(* IEC 61131-3 sources: mect_apps/AnyTPAC/TestSuite/plc (part 3) *)

(* ---- or_P.st ---- *)
(*[[ ]]*)
PROGRAM or_P
#import "Crosstable.gvl"
#import "Resource1.gvl"
CONST
	this : int := 29;
	test_cases : int := 13;
END_CONST
VAR
	test_case : array [1..test_cases] of bit2_bit_T := [
		(input0 := 0, 		    input1 := 0, 	 	   ret_bool := 0, ret_byte := 0, 	 ret_word := 0, 	ret_dword := 0),
		(input0 := 0, 			input1 := 1, 	   	   ret_bool := 1, ret_byte := 1, 	 ret_word := 1, 	ret_dword := 1),
		(input0 := 1, 			input1 := 0, 	   	   ret_bool := 1, ret_byte := 1, 	 ret_word := 1, 	ret_dword := 1),
		(input0 := 1, 			input1 := 1, 	       ret_bool := 1, ret_byte := 1, 	 ret_word := 1, 	ret_dword := 1),
		(input0 := 0, 			input1 := 16#000000ff, ret_bool := 1, ret_byte := 16#ff, ret_word := 16#00ff, ret_dword := 16#000000ff),
		(input0 := 16#000000ff, input1 := 16#000000ff, ret_bool := 1, ret_byte := 16#ff, ret_word := 16#00ff, ret_dword := 16#000000ff),
		(input0 := 16#0000000f, input1 := 16#000000f0, ret_bool := 1, ret_byte := 16#ff, ret_word := 16#00ff, ret_dword := 16#000000ff),
		(input0 := 16#0000ffff, input1 := 16#0000ffff, ret_bool := 1, ret_byte := 16#ff, ret_word := 16#ffff, ret_dword := 16#0000ffff),
		(input0 := 16#0000ffff, input1 := 16#000000ff, ret_bool := 1, ret_byte := 16#ff, ret_word := 16#ffff, ret_dword := 16#0000ffff),
		(input0 := 16#0000f000, input1 := 16#0000ffff, ret_bool := 1, ret_byte := 16#ff, ret_word := 16#ffff, ret_dword := 16#0000ffff),
		(input0 := 16#000000ff, input1 := 16#0000ff00, ret_bool := 1, ret_byte := 16#ff, ret_word := 16#ffff, ret_dword := 16#0000ffff),
		(input0 := 16#abcde012, input1 := 16#ffffffff, ret_bool := 1, ret_byte := 16#ff, ret_word := 16#ffff, ret_dword := 16#ffffffff),
		(input0 := 16#abcdefab, input1 := 16#ff000000, ret_bool := 1, ret_byte := 16#ab, ret_word := 16#efab, ret_dword := 16#ffcdefab)
	];
    ret_bool   : bool;
    ret_byte   : byte;
    ret_word   : word;
    ret_dword  : dword;

	index : int := 1;
	expected : string;
	obtained : string;
	result : bool;
END_VAR

	if Status = STATUS_RUNNING AND test_level_29 > TEST_DISABLED and test_loops_29 < Target then

		(* ---------- test action ---------------*)
        ret_bool   := or(dword_to_bool(test_case[index].input0), dword_to_bool(test_case[index].input1));
        ret_byte   := or(dword_to_byte(test_case[index].input0), dword_to_byte(test_case[index].input1));
        ret_word   := or(dword_to_word(test_case[index].input0), dword_to_word(test_case[index].input1));
        ret_dword  := or(test_case[index].input0, test_case[index].input1);

		(* ---------- test condition ---------------*)
        result := (ret_bool = test_case[index].ret_bool)
		      and (ret_byte = test_case[index].ret_byte)
		      and (ret_word = test_case[index].ret_word)
		      and (ret_dword = test_case[index].ret_dword);

		(* ---------- log message ---------------*)
		expected := '';
		expected := CONCAT(expected, comma_blank, bool_to_string(test_case[index].ret_bool));
		expected := CONCAT(expected, comma_blank, byte_to_string(test_case[index].ret_byte));
		expected := CONCAT(expected, comma_blank, word_to_string(test_case[index].ret_word));
		expected := CONCAT(expected, comma_blank, dword_to_string(test_case[index].ret_dword));
		obtained := '';
		obtained := CONCAT(obtained, comma_blank, bool_to_string(ret_bool));
		obtained := CONCAT(obtained, comma_blank, byte_to_string(ret_byte));
		obtained := CONCAT(obtained, comma_blank, word_to_string(ret_word));
		obtained := CONCAT(obtained, comma_blank, dword_to_string(ret_dword));

		(* ---------- cycle ----------*)
		SingleTest(this, result, expected, obtained, test_cases,
				   index, test_level_29, test_counter_29, test_loops_29, test_errors_29);
	end_if;
END_PROGRAM

(* ---- pow_P.st ---- *)
(*[[ ]]*)
PROGRAM pow_P
#import "Crosstable.gvl"
#import "Resource1.gvl"
CONST
	this : int := 17;
	test_cases : int := 7;
	xl : lreal := 0.0000000000000001;
	x : real := 0.0000000000000001;
END_CONST
VAR
	test_case : array [1..test_cases] of lreal_lreal4_real4_T :=
[
(input:= 0.4487989505128276, retval1:=  1.5664296956520809, retval2:=-0.8011802632059132, retval3:=-0.3479481673201230, retval4:= 0.6699245856906788, retval5:=  1.5664297018771030, retval6:=-0.8011802543511257, retval7:=-0.3479481634745377, retval8:= 0.6699245886566987),
(input:= 0.8975979010256552, retval1:=  2.4537019914206710, retval2:=-0.1080330826459679, retval3:=-0.0469181716561418, retval4:= 0.9474164348509346, retval5:=  2.4537020109227896, retval6:=-0.1080330737911804, retval7:=-0.0469181678105565, retval8:= 0.9474164390455202),
(input:= 1.3463968515384828, retval1:=  3.8435516636419869, retval2:= 0.2974320254621965, retval3:= 0.1291730873995394, retval4:= 1.1603434196557856, retval5:=  3.8435514803715054, retval6:= 0.2974319900472387, retval7:= 0.1291730720190187, retval8:= 1.1603433991090293),
(input:= 1.7951958020513104, retval1:=  6.0206534627017669, retval2:= 0.5851140979139774, retval3:= 0.2541118240078394, retval4:= 1.3398491713813576, retval5:=  6.0206535584065408, retval6:= 0.5851141067687649, retval7:= 0.2541118278534247, retval8:= 1.3398491773133974),
(input:= 2.2439947525641379, retval1:=  9.4309303712065766, retval2:= 0.8082576492281872, retval3:= 0.3510218370158958, retval4:= 1.4979969134027407, retval5:=  9.4309299964728268, retval6:= 0.8082576315211277, retval7:= 0.3510218293258176, retval8:= 1.4979969001401805),
(input:= 2.6927937030769655, retval1:= 14.7728893910850854, retval2:= 0.9905792060221418, retval3:= 0.4302030830635206, retval4:= 1.6409734010875878, retval5:= 14.7728879822659920, retval6:= 0.9905791706071840, retval7:= 0.4302030676829999, retval8:= 1.6409733720300863),
(input:= 3.1415926535897931, retval1:= 23.1406926327792668, retval2:= 1.1447298858494002, retval3:= 0.4971498726941338, retval4:= 1.7724538509055159, retval5:= 23.1406946558030384, retval6:= 1.1447299136769349, retval7:= 0.4971498847794786, retval8:= 1.7724538755670267)
];
	input_lreal : lreal;
	input_real : real;
	retval1 : lreal;
	retval2 : lreal;
	retval3 : lreal;
	retval4 : lreal;
	retval5 : real;
	retval6 : real;
	retval7 : real;
	retval8 : real;

	index : int := 1;
	expected : string;
	obtained : string;
	result : bool;
END_VAR

	if Status = STATUS_RUNNING AND test_level_17 > TEST_DISABLED and test_loops_17 < Target then

		(* ---------- test action ---------------*)
		input_lreal := test_case[index].input;
		retval1 := exp(input_lreal);
		retval2 := ln(input_lreal);
		retval3 := log(input_lreal);
		retval4 := sqrt(input_lreal);
		input_real := lreal_to_real(test_case[index].input);
		retval5 := exp(input_real);
		retval6 := ln(input_real);
		retval7 := log(input_real);
		retval8 := sqrt(input_real);

		(* ---------- test condition ---------------*)
		result := (abs(retval1 - test_case[index].retval1) < xl)
		      and (abs(retval2 - test_case[index].retval2) < xl)
		      and (abs(retval3 - test_case[index].retval3) < xl)
		      and (abs(retval4 - test_case[index].retval4) < xl)
		      and (abs(retval5 - test_case[index].retval5) < x)
		      and (abs(retval6 - test_case[index].retval6) < x)
		      and (abs(retval7 - test_case[index].retval7) < x)
		      and (abs(retval8 - test_case[index].retval8) < x);

		(* ---------- log message ---------------*)
		expected := '';
		expected := CONCAT(expected, comma_blank, lreal_to_string(test_case[index].retval1));
		expected := CONCAT(expected, comma_blank, lreal_to_string(test_case[index].retval2));
		expected := CONCAT(expected, comma_blank, lreal_to_string(test_case[index].retval3));
		expected := CONCAT(expected, comma_blank, lreal_to_string(test_case[index].retval4));
		expected := CONCAT(expected, comma_blank, real_to_string(test_case[index].retval5));
		expected := CONCAT(expected, comma_blank, real_to_string(test_case[index].retval6));
		expected := CONCAT(expected, comma_blank, real_to_string(test_case[index].retval7));
		expected := CONCAT(expected, comma_blank, real_to_string(test_case[index].retval8));
		obtained := '';
		obtained := CONCAT(obtained, comma_blank, lreal_to_string(retval1));
		obtained := CONCAT(obtained, comma_blank, lreal_to_string(retval2));
		obtained := CONCAT(obtained, comma_blank, lreal_to_string(retval3));
		obtained := CONCAT(obtained, comma_blank, lreal_to_string(retval4));
		obtained := CONCAT(obtained, comma_blank, real_to_string(retval5));
		obtained := CONCAT(obtained, comma_blank, real_to_string(retval6));
		obtained := CONCAT(obtained, comma_blank, real_to_string(retval7));
		obtained := CONCAT(obtained, comma_blank, real_to_string(retval8));

		(* ---------- cycle ----------*)
		SingleTest(this, result, expected, obtained, test_cases,
				   index, test_level_17, test_counter_17, test_loops_17, test_errors_17);
	end_if;
END_PROGRAM

(* ---- real_to_all_P.st ---- *)
(*[[
]]*)
PROGRAM real_to_all_P
#import "Crosstable.gvl"
#import "Resource1.gvl"
CONST
	this : int := 7;
	test_cases : int := 5;
END_CONST
VAR
	test_case : array [1..test_cases] of real_all_T := [
		(input := 0.0, ret_bool := 0, ret_byte := 0, ret_dword := 0, ret_int := 0, ret_dint := 0, ret_lreal := 0.0,
		   ret_string := '0', ret_time := t#0ms, ret_udint := 0, ret_uint := 0, ret_word := 0),
		(input := 1.0, ret_bool := 1, ret_byte := 1, ret_dword := 1, ret_int := 1, ret_dint := 1, ret_lreal := 1.0,
		   ret_string := '1', ret_time := t#1ms, ret_udint := 1, ret_uint := 1, ret_word := 1),
		(input := -1.0, ret_bool := 1, ret_byte := 0, ret_dword := 0, ret_int := -1, ret_dint := -1, ret_lreal := -1.0,
		   ret_string := '-1', ret_time := t#-1ms, ret_udint := 0, ret_uint := 0, ret_word := 0),
		(input := 255.0, ret_bool := 1, ret_byte := 255, ret_dword := 255, ret_int := 255, ret_dint := 255, ret_lreal := 255.0,
		   ret_string := '255', ret_time := t#255ms, ret_udint := 255, ret_uint := 255, ret_word := 255),
		(input := 400.0, ret_bool := 1, ret_byte := 255, ret_dword := 400, ret_int := 400, ret_dint := 400, ret_lreal := 400.0,
		   ret_string := '400', ret_time := t#400ms, ret_udint := 400, ret_uint := 400, ret_word := 400)
	];
    ret_bool   : bool;
    ret_byte   : byte;
    ret_dword  : dword;
    ret_int    : int;
    ret_dint   : dint;
    ret_lreal  : lreal;
    ret_string : string;
	ret_time   : time;
    ret_udint  : udint;
    ret_uint   : uint;
    ret_word   : word;

	index : int := 1;
	expected : string;
	obtained : string;
	result : bool;
END_VAR

	if Status = STATUS_RUNNING AND test_level_07 > TEST_DISABLED and test_loops_07 < Target then

		(* ---------- test action ---------------*)
        ret_bool   := real_to_bool(test_case[index].input);
        ret_byte   := real_to_byte(test_case[index].input);
        ret_dword  := real_to_dword(test_case[index].input);
        ret_int    := real_to_int(test_case[index].input);
        ret_dint   := real_to_dint(test_case[index].input);
        ret_lreal  := real_to_lreal(test_case[index].input);
        ret_string := real_to_string(test_case[index].input);
        ret_time   := real_to_time(test_case[index].input);
        ret_udint  := real_to_udint(test_case[index].input);
        ret_uint   := real_to_uint(test_case[index].input);
        ret_word   := real_to_word(test_case[index].input);

		(* ---------- test condition ---------------*)
        result := (ret_bool = test_case[index].ret_bool)
		      and (ret_byte = test_case[index].ret_byte)
		      and (ret_dword = test_case[index].ret_dword)
		      and (ret_int = test_case[index].ret_int)
		      and (ret_dint = test_case[index].ret_dint)
		      and (ret_lreal = test_case[index].ret_lreal)
		      and (ret_string = test_case[index].ret_string)
		      and (ret_time = test_case[index].ret_time)
		      and (ret_udint = test_case[index].ret_udint)
		      and (ret_uint = test_case[index].ret_uint)
		      and (ret_word = test_case[index].ret_word);

		(* ---------- log message ---------------*)
		expected := '';
		expected := CONCAT(expected, comma_blank, bool_to_string(test_case[index].ret_bool));
		expected := CONCAT(expected, comma_blank, byte_to_string(test_case[index].ret_byte));
		expected := CONCAT(expected, comma_blank, dword_to_string(test_case[index].ret_dword));
		expected := CONCAT(expected, comma_blank, int_to_string(test_case[index].ret_int));
		expected := CONCAT(expected, comma_blank, dint_to_string(test_case[index].ret_dint));
		expected := CONCAT(expected, comma_blank, lreal_to_string(test_case[index].ret_lreal));
		expected := CONCAT(expected, comma_blank, test_case[index].ret_string);
		expected := CONCAT(expected, comma_blank, time_to_string(test_case[index].ret_time));
		expected := CONCAT(expected, comma_blank, udint_to_string(test_case[index].ret_udint));
		expected := CONCAT(expected, comma_blank, uint_to_string(test_case[index].ret_uint));
		expected := CONCAT(expected, comma_blank, word_to_string(test_case[index].ret_word));
		obtained := '';
		obtained := CONCAT(obtained, comma_blank, bool_to_string(ret_bool));
		obtained := CONCAT(obtained, comma_blank, byte_to_string(ret_byte));
		obtained := CONCAT(obtained, comma_blank, dword_to_string(ret_dword));
		obtained := CONCAT(obtained, comma_blank, int_to_string(ret_int));
		obtained := CONCAT(obtained, comma_blank, dint_to_string(ret_dint));
		obtained := CONCAT(obtained, comma_blank, lreal_to_string(ret_lreal));
		obtained := CONCAT(obtained, comma_blank, ret_string);
		obtained := CONCAT(obtained, comma_blank, time_to_string(ret_time));
		obtained := CONCAT(obtained, comma_blank, udint_to_string(ret_udint));
		obtained := CONCAT(obtained, comma_blank, uint_to_string(ret_uint));
		obtained := CONCAT(obtained, comma_blank, word_to_string(ret_word));

		(* ---------- cycle ----------*)
		SingleTest(this, result, expected, obtained, test_cases,
				   index, test_level_07, test_counter_07, test_loops_07, test_errors_07);
	end_if;

END_PROGRAM

(* ---- replace_P.st ---- *)
(*[[ ]]*)
PROGRAM replace_P
#import "Crosstable.gvl"
#import "Resource1.gvl"
CONST
	this : int := 49;
	test_cases : int := 3;
END_CONST
VAR
	test_case : array [1..test_cases] of string2_int2_string_T := [
		(input0 := 'stringa_dove_inserire', input1 := 'abc_', input2 := 4,  input3 := 1,  retval := 'abc_nga_dove_inserire'),
		(input0 := 'stringa_dove_inserire', input1 := 'abc_', input2 := 4,  input3 := 8,  retval := 'stringaabc_e_inserire'),
		(input0 := 'stringa_dove_inserire', input1 := 'abc_', input2 := 4,  input3 := 21, retval := 'stringa_dove_inserirabc_')
	];
    retval0   : string;
    retval1   : string;

	index : int := 1;
	expected : string;
	obtained : string;
	result : bool;
END_VAR

	if Status = STATUS_RUNNING AND test_level_49 > TEST_DISABLED and test_loops_49 < Target then

		(* ---------- test action ---------------*)
        retval0 := replace(test_case[index].input0, test_case[index].input1, test_case[index].input2, test_case[index].input3);
        retval1 := replace(test_case[index].input0, test_case[index].input1, int_to_dint(test_case[index].input2), int_to_dint(test_case[index].input3));

		(* ---------- test condition ---------------*)
        result := (retval0 = test_case[index].retval)
		      and (retval1 = test_case[index].retval);

		(* ---------- log message ---------------*)
		expected := '';
		expected := CONCAT(expected, comma_blank, test_case[index].retval);
		expected := CONCAT(expected, comma_blank, test_case[index].retval);
		obtained := '';
		obtained := CONCAT(obtained, comma_blank, retval0);
		obtained := CONCAT(obtained, comma_blank, retval1);

		(* ---------- cycle ----------*)
		SingleTest(this, result, expected, obtained, test_cases,
				   index, test_level_49, test_counter_49, test_loops_49, test_errors_49);
	end_if;
END_PROGRAM

(* ---- ro_P.st ---- *)
(*[[ ]]*)
PROGRAM ro_P (* gestisce sia rol che ror *)
#import "Crosstable.gvl"
#import "Resource1.gvl"
CONST
	this : int := 25;
	test_cases : int := 5;
END_CONST
VAR
	test_case : array [1..test_cases] of bit2_bit2_T := [
		(input0 := 16#abcdef11, input1 := 0, ret_bool := 1, ret_byte := 16#11, ret_word := 16#ef11, ret_dword := 16#abcdef11,
											 ret_bool2 := 1, ret_byte2 := 16#11, ret_word2 := 16#ef11, ret_dword2 := 16#abcdef11),
		(input0 := 16#abcdef11, input1 := 1, ret_bool := 1, ret_byte := 16#22, ret_word := 16#de23, ret_dword := 16#579bde23,
											 ret_bool2 := 1, ret_byte2 := 16#88, ret_word2 := 16#f788, ret_dword2 := 16#d5e6f788),
		(input0 := 16#abcdef12, input1 := 2, ret_bool := 1, ret_byte := 16#48, ret_word := 16#bc4b, ret_dword := 16#af37bc4a,
											 ret_bool2 := 1, ret_byte2 := 16#84, ret_word2 := 16#bbc4, ret_dword2 := 16#aaf37bc4),
		(input0 := 16#abcdef12, input1 := 4, ret_bool := 1, ret_byte := 16#21, ret_word := 16#f12e, ret_dword := 16#bcdef12a,
											 ret_bool2 := 1, ret_byte2 := 16#21, ret_word2 := 16#2ef1, ret_dword2 := 16#2abcdef1),
		(input0 := 16#abcdef12, input1 := 7, ret_bool := 1, ret_byte := 16#09, ret_word := 16#8977, ret_dword := 16#e6f78955,
											 ret_bool2 := 1, ret_byte2 := 16#24, ret_word2 := 16#25de, ret_dword2 := 16#25579bde)
	];
    ret_bool   : bool;
    ret_byte   : byte;
    ret_word   : word;
    ret_dword  : dword;
    ret_bool2  : bool;
    ret_byte2  : byte;
    ret_word2  : word;
    ret_dword2 : dword;

	index : int := 1;
	expected : string;
	obtained : string;
	result : bool;
END_VAR

	if Status = STATUS_RUNNING AND test_level_25 > TEST_DISABLED and test_loops_25 < Target then

		(* ---------- test action ---------------*)
        ret_bool   := rol(dword_to_bool(test_case[index].input0), dword_to_int(test_case[index].input1));
        ret_byte   := rol(dword_to_byte(test_case[index].input0), dword_to_int(test_case[index].input1));
        ret_word   := rol(dword_to_word(test_case[index].input0), dword_to_int(test_case[index].input1));
        ret_dword  := rol(test_case[index].input0, dword_to_int(test_case[index].input1));
        ret_bool2  := ror(dword_to_bool(test_case[index].input0), dword_to_int(test_case[index].input1));
        ret_byte2  := ror(dword_to_byte(test_case[index].input0), dword_to_int(test_case[index].input1));
        ret_word2  := ror(dword_to_word(test_case[index].input0), dword_to_int(test_case[index].input1));
        ret_dword2 := ror(test_case[index].input0, dword_to_int(test_case[index].input1));

		(* ---------- test condition ---------------*)
        result := (ret_bool = test_case[index].ret_bool)
		      and (ret_byte = test_case[index].ret_byte)
		      and (ret_word = test_case[index].ret_word)
		      and (ret_dword = test_case[index].ret_dword)
			  and (ret_bool2 = test_case[index].ret_bool2)
		      and (ret_byte2 = test_case[index].ret_byte2)
		      and (ret_word2 = test_case[index].ret_word2)
		      and (ret_dword2 = test_case[index].ret_dword2);

		(* ---------- log message ---------------*)
		expected := '';
		expected := CONCAT(expected, comma_blank, bool_to_string(test_case[index].ret_bool));
		expected := CONCAT(expected, comma_blank, byte_to_string(test_case[index].ret_byte));
		expected := CONCAT(expected, comma_blank, word_to_string(test_case[index].ret_word));
		expected := CONCAT(expected, comma_blank, dword_to_string(test_case[index].ret_dword));
		expected := CONCAT(expected, comma_blank, bool_to_string(test_case[index].ret_bool2));
		expected := CONCAT(expected, comma_blank, byte_to_string(test_case[index].ret_byte2));
		expected := CONCAT(expected, comma_blank, word_to_string(test_case[index].ret_word2));
		expected := CONCAT(expected, comma_blank, dword_to_string(test_case[index].ret_dword2));
		obtained := '';
		obtained := CONCAT(obtained, comma_blank, bool_to_string(ret_bool));
		obtained := CONCAT(obtained, comma_blank, byte_to_string(ret_byte));
		obtained := CONCAT(obtained, comma_blank, word_to_string(ret_word));
		obtained := CONCAT(obtained, comma_blank, dword_to_string(ret_dword));
		obtained := CONCAT(obtained, comma_blank, bool_to_string(ret_bool2));
		obtained := CONCAT(obtained, comma_blank, byte_to_string(ret_byte2));
		obtained := CONCAT(obtained, comma_blank, word_to_string(ret_word2));
		obtained := CONCAT(obtained, comma_blank, dword_to_string(ret_dword2));

		(* ---------- cycle ----------*)
		SingleTest(this, result, expected, obtained, test_cases,
				   index, test_level_25, test_counter_25, test_loops_25, test_errors_25);
	end_if;
END_PROGRAM

(* ---- rs_sr_P.st ---- *)
(*[[
]]*)
PROGRAM rs_sr_P
#import "Crosstable.gvl"
#import "Resource1.gvl"
CONST
	this : int := 52;
	test_cases : int := 11;
END_CONST
VAR
	test_case : array [1..test_cases] of bool2_bool2_T := [

		(input1 := false, input2 := false, retval1 := false, retval2 := false),
		(input1 := true,  input2 := false, retval1 := true,  retval2 := true),
		(input1 := false, input2 := false, retval1 := true,  retval2 := true),

		(input1 := false, input2 := false, retval1 := true,  retval2 := true),
		(input1 := false, input2 := true,  retval1 := false, retval2 := false),
		(input1 := false, input2 := false, retval1 := false, retval2 := false),

		(input1 := true,  input2 := true,  retval1 := false, retval2 := true),
		(input1 := false, input2 := false, retval1 := false, retval2 := true),
		(input1 := false, input2 := false, retval1 := false, retval2 := true),

		(input1 := false, input2 := true,  retval1 := false, retval2 := false),
		(input1 := false, input2 := false, retval1 := false, retval2 := false)
		];

    retval1  : bool;
    retval2  : bool;

	RS_Inst : RS;
	SR_Inst : SR;
	index : int := 1;
	expected : string;
	obtained : string;
	result : bool;
END_VAR

	if Status = STATUS_RUNNING AND test_level_52 > TEST_DISABLED and test_loops_52 < Target then

		(* ---------- test action ---------------*)
		RS_Inst(S := test_case[index].input1, R1 := test_case[index].input2, Q1 => retval1);
		SR_Inst(S1 := test_case[index].input1, R := test_case[index].input2, Q1 => retval2);

		(* ---------- test condition ---------------*)
        result := (retval1 = test_case[index].retval1)
		      and (retval2 = test_case[index].retval2);

		(* ---------- log message ---------------*)
		expected := '';
		expected := CONCAT(expected, comma_blank, bool_to_string(test_case[index].retval1));
		expected := CONCAT(expected, comma_blank, bool_to_string(test_case[index].retval2));
		obtained := '';
		obtained := CONCAT(obtained, comma_blank, bool_to_string(retval1));
		obtained := CONCAT(obtained, comma_blank, bool_to_string(retval2));

		(* ---------- cycle ----------*)
		SingleTest(this, result, expected, obtained, test_cases,
				   index, test_level_52, test_counter_52, test_loops_52, test_errors_52);
	end_if;
END_PROGRAM

(* ---- sel_P.st ---- *)
(*[[ ]]*)
PROGRAM sel_P
#import "Crosstable.gvl"
#import "Resource1.gvl"
CONST
	this : int := 35;
	test_cases : int := 2;
END_CONST
VAR
	test_case : array [1..test_cases] of bool_any2_any_T := [
		(input0 := false,  input1 := 20.0,  input2 := 30.0,  ret_byte := 20, ret_word := 20, ret_dword := 20, ret_int := 20, ret_dint := 20,
															ret_time := t#20ms, ret_real := 20.0, ret_lreal := 20.0, ret_string := '20'),
		(input0 := true,  input1 := 10.0,  input2 := 20.0,  ret_byte := 20, ret_word := 20, ret_dword := 20, ret_int := 20, ret_dint := 20,
															ret_time := t#20ms, ret_real := 20.0, ret_lreal := 20.0, ret_string := '20')
	];
    ret_byte   : byte;
    ret_word   : word;
    ret_dword  : dword;
    ret_int    : int;
    ret_dint   : dint;
    ret_time   : time;
    ret_real   : real;
    ret_lreal  : lreal;
    ret_string : string;

	index : int := 1;
	expected : string;
	obtained : string;
	result : bool;
END_VAR

	if Status = STATUS_RUNNING AND test_level_35 > TEST_DISABLED and test_loops_35 < Target then

		(* ---------- test action ---------------*)
        ret_byte    := sel(test_case[index].input0, lreal_to_byte(test_case[index].input1), lreal_to_byte(test_case[index].input2));
        ret_word    := sel(test_case[index].input0, lreal_to_word(test_case[index].input1), lreal_to_word(test_case[index].input2));
        ret_dword   := sel(test_case[index].input0, lreal_to_dword(test_case[index].input1), lreal_to_dword(test_case[index].input2));
        ret_int     := sel(test_case[index].input0, lreal_to_int(test_case[index].input1), lreal_to_int(test_case[index].input2));
        ret_dint    := sel(test_case[index].input0, lreal_to_dint(test_case[index].input1), lreal_to_dint(test_case[index].input2));
        ret_time    := sel(test_case[index].input0, lreal_to_time(test_case[index].input1), lreal_to_time(test_case[index].input2));
        ret_real    := sel(test_case[index].input0, lreal_to_real(test_case[index].input1), lreal_to_real(test_case[index].input2));
        ret_lreal   := sel(test_case[index].input0, test_case[index].input1, test_case[index].input2);
        ret_string  := sel(test_case[index].input0, lreal_to_string(test_case[index].input1), lreal_to_string(test_case[index].input2));

		(* ---------- test condition ---------------*)
        result := ((ret_byte = test_case[index].ret_byte)
			  and (ret_word = test_case[index].ret_word)
			  and (ret_dword = test_case[index].ret_dword)
			  and (ret_int = test_case[index].ret_int)
		      and (ret_dint = test_case[index].ret_dint)
		      and (ret_time = test_case[index].ret_time)
		      and (ret_real = test_case[index].ret_real)
		      and (ret_lreal = test_case[index].ret_lreal)
		      and (ret_string = test_case[index].ret_string));

		(* ---------- log message ---------------*)
		expected := '';
		expected := CONCAT(expected, comma_blank, byte_to_string(test_case[index].ret_byte));
		expected := CONCAT(expected, comma_blank, word_to_string(test_case[index].ret_word));
		expected := CONCAT(expected, comma_blank, dword_to_string(test_case[index].ret_dword));
		expected := CONCAT(expected, comma_blank, int_to_string(test_case[index].ret_int));
		expected := CONCAT(expected, comma_blank, dint_to_string(test_case[index].ret_dint));
		expected := CONCAT(expected, comma_blank, time_to_string(test_case[index].ret_time));
		expected := CONCAT(expected, comma_blank, real_to_string(test_case[index].ret_real));
		expected := CONCAT(expected, comma_blank, lreal_to_string(test_case[index].ret_lreal));
		expected := CONCAT(expected, comma_blank, test_case[index].ret_string);
		obtained := '';
		obtained := CONCAT(obtained, comma_blank, byte_to_string(ret_byte));
		obtained := CONCAT(obtained, comma_blank, word_to_string(ret_word));
		obtained := CONCAT(obtained, comma_blank, dword_to_string(ret_dword));
		obtained := CONCAT(obtained, comma_blank, int_to_string(ret_int));
		obtained := CONCAT(obtained, comma_blank, dint_to_string(ret_dint));
		obtained := CONCAT(obtained, comma_blank, time_to_string(ret_time));
		obtained := CONCAT(obtained, comma_blank, real_to_string(ret_real));
		obtained := CONCAT(obtained, comma_blank, lreal_to_string(ret_lreal));
		obtained := CONCAT(obtained, comma_blank, ret_string);

		(* ---------- cycle ----------*)
		SingleTest(this, result, expected, obtained, test_cases,
				   index, test_level_35, test_counter_35, test_loops_35, test_errors_35);
	end_if;
END_PROGRAM

(* ---- sh_P.st ---- *)
(*[[ ]]*)
PROGRAM sh_P (* gestisce sia shl che shr *)
#import "Crosstable.gvl"
#import "Resource1.gvl"
CONST
	this : int := 26;
	test_cases : int := 5;
END_CONST
VAR
	test_case : array [1..test_cases] of bit2_bit2_T := [
		(input0 := 16#abcdef11, input1 := 0, ret_bool := 1, ret_byte := 16#11, ret_word := 16#ef11, ret_dword := 16#abcdef11,
											 ret_bool2 := 1, ret_byte2 := 16#11, ret_word2 := 16#ef11, ret_dword2 := 16#abcdef11),
		(input0 := 16#abcdef11, input1 := 1, ret_bool := 0, ret_byte := 16#22, ret_word := 16#de22, ret_dword := 16#579bde22,
											 ret_bool2 := 0, ret_byte2 := 16#08, ret_word2 := 16#7788, ret_dword2 := 16#55e6f788),
		(input0 := 16#abcdef12, input1 := 2, ret_bool := 0, ret_byte := 16#48, ret_word := 16#bc48, ret_dword := 16#af37bc48,
											 ret_bool2 := 0, ret_byte2 := 16#04, ret_word2 := 16#3bc4, ret_dword2 := 16#2af37bc4),
		(input0 := 16#abcdef12, input1 := 4, ret_bool := 0, ret_byte := 16#20, ret_word := 16#f120, ret_dword := 16#bcdef120,
											 ret_bool2 := 0, ret_byte2 := 16#01, ret_word2 := 16#0ef1, ret_dword2 := 16#0abcdef1),
		(input0 := 16#abcdef12, input1 := 7, ret_bool := 0, ret_byte := 16#00, ret_word := 16#8900, ret_dword := 16#e6f78900,
											 ret_bool2 := 0, ret_byte2 := 16#00, ret_word2 := 16#01de, ret_dword2 := 16#01579bde)
	];
    ret_bool   : bool;
    ret_byte   : byte;
    ret_word   : word;
    ret_dword  : dword;
    ret_bool2  : bool;
    ret_byte2  : byte;
    ret_word2  : word;
    ret_dword2 : dword;

	index : int := 1;
	expected : string;
	obtained : string;
	result : bool;
END_VAR

	if Status = STATUS_RUNNING AND test_level_26 > TEST_DISABLED and test_loops_26 < Target then

		(* ---------- test action ---------------*)
        ret_bool   := shl(dword_to_bool(test_case[index].input0), dword_to_int(test_case[index].input1));
        ret_byte   := shl(dword_to_byte(test_case[index].input0), dword_to_int(test_case[index].input1));
        ret_word   := shl(dword_to_word(test_case[index].input0), dword_to_int(test_case[index].input1));
        ret_dword  := shl(test_case[index].input0, dword_to_int(test_case[index].input1));
        ret_bool2  := shr(dword_to_bool(test_case[index].input0), dword_to_int(test_case[index].input1));
        ret_byte2  := shr(dword_to_byte(test_case[index].input0), dword_to_int(test_case[index].input1));
        ret_word2  := shr(dword_to_word(test_case[index].input0), dword_to_int(test_case[index].input1));
        ret_dword2 := shr(test_case[index].input0, dword_to_int(test_case[index].input1));

		(* ---------- test condition ---------------*)
        result := (ret_bool = test_case[index].ret_bool)
		      and (ret_byte = test_case[index].ret_byte)
		      and (ret_word = test_case[index].ret_word)
		      and (ret_dword = test_case[index].ret_dword)
			  and (ret_bool2 = test_case[index].ret_bool2)
		      and (ret_byte2 = test_case[index].ret_byte2)
		      and (ret_word2 = test_case[index].ret_word2)
		      and (ret_dword2 = test_case[index].ret_dword2);

		(* ---------- log message ---------------*)
		expected := '';
		expected := CONCAT(expected, comma_blank, bool_to_string(test_case[index].ret_bool));
		expected := CONCAT(expected, comma_blank, byte_to_string(test_case[index].ret_byte));
		expected := CONCAT(expected, comma_blank, word_to_string(test_case[index].ret_word));
		expected := CONCAT(expected, comma_blank, dword_to_string(test_case[index].ret_dword));
		expected := CONCAT(expected, comma_blank, bool_to_string(test_case[index].ret_bool2));
		expected := CONCAT(expected, comma_blank, byte_to_string(test_case[index].ret_byte2));
		expected := CONCAT(expected, comma_blank, word_to_string(test_case[index].ret_word2));
		expected := CONCAT(expected, comma_blank, dword_to_string(test_case[index].ret_dword2));
		obtained := '';
		obtained := CONCAT(obtained, comma_blank, bool_to_string(ret_bool));
		obtained := CONCAT(obtained, comma_blank, byte_to_string(ret_byte));
		obtained := CONCAT(obtained, comma_blank, word_to_string(ret_word));
		obtained := CONCAT(obtained, comma_blank, dword_to_string(ret_dword));
		obtained := CONCAT(obtained, comma_blank, bool_to_string(ret_bool2));
		obtained := CONCAT(obtained, comma_blank, byte_to_string(ret_byte2));
		obtained := CONCAT(obtained, comma_blank, word_to_string(ret_word2));
		obtained := CONCAT(obtained, comma_blank, dword_to_string(ret_dword2));

		(* ---------- cycle ----------*)
		SingleTest(this, result, expected, obtained, test_cases,
				   index, test_level_26, test_counter_26, test_loops_26, test_errors_26);
	end_if;
END_PROGRAM

(* ---- string_to_all_P.st ---- *)
(*[[
]]*)
PROGRAM string_to_all_P
#import "Crosstable.gvl"
#import "Resource1.gvl"
CONST
	this : int := 8;
	test_cases : int := 5;
END_CONST
VAR
	test_case : array [1..test_cases] of string_all_T := [
		(input := '0', ret_bool := 0, ret_byte := 0, ret_dword := 0, ret_int := 0, ret_dint := 0, ret_lreal := 0.0,
		   ret_real := 0.0, ret_time := t#0ms, ret_udint := 0, ret_uint := 0, ret_word := 0),
		(input := '1', ret_bool := 1, ret_byte := 1, ret_dword := 1, ret_int := 1, ret_dint := 1, ret_lreal := 1.0,
		   ret_real := 1.0, ret_time := t#1ms, ret_udint := 1, ret_uint := 1, ret_word := 1),
		(input := '-1', ret_bool := 0, ret_byte := 255, ret_dword := 16#ffffffff, ret_int := -1, ret_dint := -1, ret_lreal := -1.0,
		   ret_real := -1.0, ret_time := t#-1ms, ret_udint := 16#ffffffff, ret_uint := 16#ffff, ret_word := 16#ffff),
		(input := '255', ret_bool := 0, ret_byte := 255, ret_dword := 255, ret_int := 255, ret_dint := 255, ret_lreal := 255.0,
		   ret_real := 255.0, ret_time := t#255ms, ret_udint := 255, ret_uint := 255, ret_word := 255),
		(input := '400', ret_bool := 0, ret_byte := 144, ret_dword := 400, ret_int := 400, ret_dint := 400, ret_lreal := 400.0,
		   ret_real := 400.0, ret_time := t#400ms, ret_udint := 400, ret_uint := 400, ret_word := 400)
	];
    ret_bool   : bool;
    ret_byte   : byte;
    ret_dword  : dword;
    ret_int    : int;
    ret_dint   : dint;
    ret_lreal  : lreal;
    ret_real   : real;
    ret_time   : time;
    ret_udint  : udint;
    ret_uint   : uint;
    ret_word   : word;

	index : int := 1;
	expected : string;
	obtained : string;
	result : bool;
END_VAR

	if Status = STATUS_RUNNING AND test_level_08 > TEST_DISABLED and test_loops_08 < Target then

		(* ---------- test action ---------------*)
        ret_bool   := string_to_bool(test_case[index].input);
        ret_byte   := string_to_byte(test_case[index].input);
        ret_dword  := string_to_dword(test_case[index].input);
        ret_int    := string_to_int(test_case[index].input);
        ret_dint   := string_to_dint(test_case[index].input);
        ret_lreal  := string_to_lreal(test_case[index].input);
        ret_real   := string_to_real(test_case[index].input);
        ret_time   := string_to_time(concat('t#', test_case[index].input, 'ms'));
        ret_udint  := string_to_udint(test_case[index].input);
        ret_uint   := string_to_uint(test_case[index].input);
        ret_word   := string_to_word(test_case[index].input);

		(* ---------- test condition ---------------*)
        result := (ret_bool = test_case[index].ret_bool)
		      and (ret_byte = test_case[index].ret_byte)
		      and (ret_dword = test_case[index].ret_dword)
		      and (ret_int = test_case[index].ret_int)
		      and (ret_dint = test_case[index].ret_dint)
		      and (ret_lreal = test_case[index].ret_lreal)
		      and (ret_real = test_case[index].ret_real)
		      and (ret_time = test_case[index].ret_time)
		      and (ret_udint = test_case[index].ret_udint)
		      and (ret_uint = test_case[index].ret_uint)
		      and (ret_word = test_case[index].ret_word);

		(* ---------- log message ---------------*)
		expected := '';
		expected := CONCAT(expected, comma_blank, bool_to_string(test_case[index].ret_bool));
		expected := CONCAT(expected, comma_blank, byte_to_string(test_case[index].ret_byte));
		expected := CONCAT(expected, comma_blank, dword_to_string(test_case[index].ret_dword));
		expected := CONCAT(expected, comma_blank, int_to_string(test_case[index].ret_int));
		expected := CONCAT(expected, comma_blank, dint_to_string(test_case[index].ret_dint));
		expected := CONCAT(expected, comma_blank, lreal_to_string(test_case[index].ret_lreal));
		expected := CONCAT(expected, comma_blank, real_to_string(test_case[index].ret_real));
		expected := CONCAT(expected, comma_blank, time_to_string(test_case[index].ret_time));
		expected := CONCAT(expected, comma_blank, udint_to_string(test_case[index].ret_udint));
		expected := CONCAT(expected, comma_blank, uint_to_string(test_case[index].ret_uint));
		expected := CONCAT(expected, comma_blank, word_to_string(test_case[index].ret_word));
		obtained := '';
		obtained := CONCAT(obtained, comma_blank, bool_to_string(ret_bool));
		obtained := CONCAT(obtained, comma_blank, byte_to_string(ret_byte));
		obtained := CONCAT(obtained, comma_blank, dword_to_string(ret_dword));
		obtained := CONCAT(obtained, comma_blank, int_to_string(ret_int));
		obtained := CONCAT(obtained, comma_blank, dint_to_string(ret_dint));
		obtained := CONCAT(obtained, comma_blank, lreal_to_string(ret_lreal));
		obtained := CONCAT(obtained, comma_blank, real_to_string(ret_real));
		obtained := CONCAT(obtained, comma_blank, time_to_string(ret_time));
		obtained := CONCAT(obtained, comma_blank, udint_to_string(ret_udint));
		obtained := CONCAT(obtained, comma_blank, uint_to_string(ret_uint));
		obtained := CONCAT(obtained, comma_blank, word_to_string(ret_word));

		(* ---------- cycle ----------*)
		SingleTest(this, result, expected, obtained, test_cases,
				   index, test_level_08, test_counter_08, test_loops_08, test_errors_08);
	end_if;

END_PROGRAM

(* ---- sub_P.st ---- *)
(*[[ ]]*)
PROGRAM sub_P
#import "Crosstable.gvl"
#import "Resource1.gvl"
CONST
	this : int := 24;
	test_cases : int := 4;
END_CONST
VAR
	test_case : array [1..test_cases] of num2_num_T := [
		(input0 := 10.0, input1 := 10.0, ret_int := 0, ret_dint := 0, ret_udint := 0, ret_uint := 0, ret_real := 0.0, ret_lreal := 0.0),
		(input0 := 10.0, input1 := 100.0, ret_int := -90, ret_dint := -90, ret_udint := 4294967206, ret_uint := 65446, ret_real := -90.0, ret_lreal := -90.0),
		(input0 := 100.0, input1 := 10.0, ret_int := 90, ret_dint := 90, ret_udint := 90, ret_uint := 90, ret_real := 90.0, ret_lreal := 90.0),
		(input0 := -10.0, input1 := -40.0, ret_int := 30, ret_dint := 30, ret_udint := 0, ret_uint := 0, ret_real := 30.0, ret_lreal := 30.0)
	];
    ret_int    : int;
    ret_dint   : dint;
    ret_uint   : uint;
    ret_udint  : udint;
    ret_real   : real;
    ret_lreal  : lreal;

	index : int := 1;
	expected : string;
	obtained : string;
	result : bool;
END_VAR

	if Status = STATUS_RUNNING AND test_level_24 > TEST_DISABLED and test_loops_24 < Target then

		(* ---------- test action ---------------*)
        ret_int     := sub(lreal_to_int(test_case[index].input0), lreal_to_int(test_case[index].input1));
        ret_dint    := sub(lreal_to_dint(test_case[index].input0), lreal_to_dint(test_case[index].input1));
        ret_uint    := sub(lreal_to_uint(test_case[index].input0), lreal_to_uint(test_case[index].input1));
        ret_udint   := sub(lreal_to_udint(test_case[index].input0), lreal_to_udint(test_case[index].input1));
        ret_real    := sub(lreal_to_real(test_case[index].input0), lreal_to_real(test_case[index].input1));
        ret_lreal   := sub(test_case[index].input0, test_case[index].input1);

		(* ---------- test condition ---------------*)
        result := ((ret_int = test_case[index].ret_int)
		      and (ret_dint = test_case[index].ret_dint)
		      and (ret_uint = test_case[index].ret_uint)
		      and (ret_udint = test_case[index].ret_udint)
		      and (ret_real = test_case[index].ret_real)
		      and (ret_lreal = test_case[index].ret_lreal));

		(* ---------- log message ---------------*)
		expected := '';
		expected := CONCAT(expected, comma_blank, int_to_string(test_case[index].ret_int));
		expected := CONCAT(expected, comma_blank, dint_to_string(test_case[index].ret_dint));
		expected := CONCAT(expected, comma_blank, uint_to_string(test_case[index].ret_uint));
		expected := CONCAT(expected, comma_blank, udint_to_string(test_case[index].ret_udint));
		expected := CONCAT(expected, comma_blank, real_to_string(test_case[index].ret_real));
		expected := CONCAT(expected, comma_blank, lreal_to_string(test_case[index].ret_lreal));
		obtained := '';
		obtained := CONCAT(obtained, comma_blank, int_to_string(ret_int));
		obtained := CONCAT(obtained, comma_blank, dint_to_string(ret_dint));
		obtained := CONCAT(obtained, comma_blank, uint_to_string(ret_uint));
		obtained := CONCAT(obtained, comma_blank, udint_to_string(ret_udint));
		obtained := CONCAT(obtained, comma_blank, real_to_string(ret_real));
		obtained := CONCAT(obtained, comma_blank, lreal_to_string(ret_lreal));

		(* ---------- cycle ----------*)
		SingleTest(this, result, expected, obtained, test_cases,
				   index, test_level_24, test_counter_24, test_loops_24, test_errors_24);
	end_if;
END_PROGRAM

(* ---- time_to_all_P.st ---- *)
(*[[
]]*)
PROGRAM time_to_all_P
#import "Crosstable.gvl"
#import "Resource1.gvl"
CONST
	this : int := 9;
	test_cases : int := 5;
END_CONST
VAR
	test_case : array [1..test_cases] of time_all_T := [
		(input := t#0ms, ret_dint := 0,  ret_int := 0, ret_lreal := 0.0, ret_real := 0.0, ret_string := 't#0ms'),
		(input := t#1ms, ret_dint := 1, ret_int := 1, ret_lreal := 1.0, ret_real := 1.0, ret_string := 't#1ms'),
		(input := t#-1ms, ret_dint := -1, ret_int := -1, ret_lreal := -1.0, ret_real := -1.0, ret_string := 't#-1ms'),
		(input := t#255ms, ret_dint := 255, ret_int := 255, ret_lreal := 255.0, ret_real := 255.0, ret_string := 't#255ms'),
		(input := t#400ms, ret_dint := 400, ret_int := 400, ret_lreal := 400.0, ret_real := 400.0, ret_string := 't#400ms')
	];
    ret_dint   : dint;
    ret_int    : int;
    ret_lreal  : lreal;
    ret_real   : real;
    ret_string : string;

	index : int := 1;
	expected: string;
	obtained: string;
	result : bool;
END_VAR

	if Status = STATUS_RUNNING AND test_level_09 > TEST_DISABLED and test_loops_09 < Target then

		(* ---------- test action ---------------*)
        ret_dint   := time_to_dint(test_case[index].input);
        ret_int    := time_to_int(test_case[index].input);
        ret_lreal  := time_to_lreal(test_case[index].input);
        ret_real   := time_to_real(test_case[index].input);
        ret_string := time_to_string(test_case[index].input);

		(* ---------- test condition ---------------*)
        result := (ret_dint = test_case[index].ret_dint)
		      and (ret_int = test_case[index].ret_int)
		      and (ret_lreal = test_case[index].ret_lreal)
		      and (ret_real = test_case[index].ret_real)
		      and (ret_string = test_case[index].ret_string);

		(* ---------- log message ---------------*)
		expected := '';
		expected := CONCAT(expected, comma_blank, dint_to_string(test_case[index].ret_dint));
		expected := CONCAT(expected, comma_blank, int_to_string(test_case[index].ret_int));
		expected := CONCAT(expected, comma_blank, lreal_to_string(test_case[index].ret_lreal));
		expected := CONCAT(expected, comma_blank, real_to_string(test_case[index].ret_real));
		expected := CONCAT(expected, comma_blank, test_case[index].ret_string);
		obtained := '';
		obtained := CONCAT(obtained, comma_blank, dint_to_string(ret_dint));
		obtained := CONCAT(obtained, comma_blank, int_to_string(ret_int));
		obtained := CONCAT(obtained, comma_blank, lreal_to_string(ret_lreal));
		obtained := CONCAT(obtained, comma_blank, real_to_string(ret_real));
		obtained := CONCAT(obtained, comma_blank, ret_string);

		(* ---------- cycle ----------*)
		SingleTest(this, result, expected, obtained, test_cases,
				   index, test_level_09, test_counter_09, test_loops_09, test_errors_09);
	end_if;
END_PROGRAM

(* ---- tof_ton_tp_P.st ---- *)
(*[[
]]*)
PROGRAM tof_ton_tp_P
#import "Crosstable.gvl"
#import "Resource1.gvl"
CONST
	this : int := 55;
	test_cases : int := 16;
END_CONST
VAR
	test_case : array [1..test_cases] of bool_time_bool3_time3_T := [

		(* reset all_____________________   TP______________________________  TON_____________________________  TOF_____________________________ *)
		(bool0 := false, time0 := t#000ms,  bool1 := false, time1 := t#000ms, bool2 := false, time2 := t#000ms, bool3 := false, time3 := t#000ms),

		(* start, reset TON, wait TP+TOF_   TP______________________________  TON_____________________________  TOF_____________________________ *)
		(bool0 := true,  time0 := t#250ms,  bool1 := true,  time1 := t#000ms, bool2 := false, time2 := t#000ms, bool3 := true,  time3 := t#000ms),
		(bool0 := false, time0 := t#250ms,  bool1 := true,  time1 := t#100ms, bool2 := false, time2 := t#000ms, bool3 := true,  time3 := t#000ms),
		(bool0 := false, time0 := t#250ms,  bool1 := true,  time1 := t#200ms, bool2 := false, time2 := t#000ms, bool3 := true,  time3 := t#100ms),
		(bool0 := false, time0 := t#250ms,  bool1 := false, time1 := t#000ms, bool2 := false, time2 := t#000ms, bool3 := true,  time3 := t#200ms),
		(bool0 := false, time0 := t#250ms,  bool1 := false, time1 := t#000ms, bool2 := false, time2 := t#000ms, bool3 := false, time3 := t#250ms),

		(* reset all_____________________   TP______________________________  TON_____________________________  TOF_____________________________ *)
		(bool0 := false, time0 := t#000ms,  bool1 := false, time1 := t#000ms, bool2 := false, time2 := t#000ms, bool3 := false, time3 := t#000ms),

		(* start and wait TP+TON_________   TP______________________________  TON_____________________________  TOF_____________________________ *)
		(bool0 := true,  time0 := t#250ms,  bool1 := true,  time1 := t#000ms, bool2 := false, time2 := t#000ms, bool3 := true,  time3 := t#000ms),
		(bool0 := true,  time0 := t#250ms,  bool1 := true,  time1 := t#100ms, bool2 := false, time2 := t#100ms, bool3 := true,  time3 := t#000ms),
		(bool0 := true,  time0 := t#250ms,  bool1 := true,  time1 := t#200ms, bool2 := false, time2 := t#200ms, bool3 := true,  time3 := t#000ms),
		(bool0 := true,  time0 := t#250ms,  bool1 := false, time1 := t#250ms, bool2 := true,  time2 := t#250ms, bool3 := true,  time3 := t#000ms),

		(* reset all_____________________   TP______________________________  TON_____________________________  TOF_____________________________ *)
		(bool0 := false, time0 := t#250ms,  bool1 := false, time1 := t#000ms, bool2 := false, time2 := t#000ms, bool3 := true,  time3 := t#000ms),

		(* start and wait TOF____________   TP______________________________  TON_____________________________  TOF_____________________________ *)
		(bool0 := false, time0 := t#250ms,  bool1 := false, time1 := t#000ms, bool2 := false, time2 := t#000ms, bool3 := true,  time3 := t#100ms),
		(bool0 := false, time0 := t#250ms,  bool1 := false, time1 := t#000ms, bool2 := false, time2 := t#000ms, bool3 := true,  time3 := t#200ms),
		(bool0 := false, time0 := t#250ms,  bool1 := false, time1 := t#000ms, bool2 := false, time2 := t#000ms, bool3 := false, time3 := t#250ms),

		(* reset all_____________________   TP______________________________  TON_____________________________  TOF_____________________________ *)
		(bool0 := false, time0 := t#000ms,  bool1 := false, time1 := t#000ms, bool2 := false, time2 := t#000ms, bool3 := false, time3 := t#000ms)
	];

    bool1, bool2, bool3 : bool;
    time1, time2, time3 : time;
	delta1, delta2, delta3: dint;

	TP_Inst : TP;
	TON_Inst : TON;
	TOF_Inst : TOF;
	index : int := 1;
	expected : string;
	obtained : string;
	result : bool;
	period_ms : time;
	info : tsk_info;
	retval : word;
END_VAR

	if Status = STATUS_RUNNING AND test_level_55 > TEST_DISABLED and test_loops_55 < Target then

		retval := TSK_GetInfo(TSK_GetMyName(), info);
		period_ms := info.tCycle;
		if period_ms <> t#100ms then
			MSG_SendToEng('ERROR: Program TOF_TON_TP must run @ 100ms: disabled.');
			test_level_55 := 0;
			return;
		end_if;

		(* ---------- test action ---------------*)
		TP_Inst (IN := test_case[index].bool0, PT := test_case[index].time0, Q => bool1, ET => time1);
		TON_Inst(IN := test_case[index].bool0, PT := test_case[index].time0, Q => bool2, ET => time2);
		TOF_Inst(IN := test_case[index].bool0, PT := test_case[index].time0, Q => bool3, ET => time3);

		delta1 := time_to_dint(time1 - test_case[index].time1);
		delta2 := time_to_dint(time2 - test_case[index].time2);
		delta3 := time_to_dint(time3 - test_case[index].time3);

		(* ---------- test condition ---------------*)
        result := (bool1 = test_case[index].bool1) and (abs(delta1) < 10)
		      and (bool2 = test_case[index].bool2) and (abs(delta2) < 10)
		      and (bool3 = test_case[index].bool3) and (abs(delta3) < 10);

		(* ---------- log message ---------------*)
		expected := '';
		expected := CONCAT(expected, comma_blank, bool_to_string(test_case[index].bool1));
		expected := CONCAT(expected, comma_blank, time_to_string(test_case[index].time1));
		expected := CONCAT(expected, comma_blank, bool_to_string(test_case[index].bool2));
		expected := CONCAT(expected, comma_blank, time_to_string(test_case[index].time2));
		expected := CONCAT(expected, comma_blank, bool_to_string(test_case[index].bool3));
		expected := CONCAT(expected, comma_blank, time_to_string(test_case[index].time3));
		obtained := '';
		obtained := CONCAT(obtained, comma_blank, bool_to_string(bool1));
		obtained := CONCAT(obtained, comma_blank, time_to_string(time1));
		obtained := CONCAT(obtained, comma_blank, bool_to_string(bool2));
		obtained := CONCAT(obtained, comma_blank, time_to_string(time2));
		obtained := CONCAT(obtained, comma_blank, bool_to_string(bool3));
		obtained := CONCAT(obtained, comma_blank, time_to_string(time3));

		(* ---------- cycle ----------*)
		if not result then
			;
		end_if;
		SingleTest(this, result, expected, obtained, test_cases,
				   index, test_level_55, test_counter_55, test_loops_55, test_errors_55);
	end_if;
END_PROGRAM

(* ---- trig_inv_P.st ---- *)
(*[[ ]]*)
PROGRAM trig_inv_P
#import "Crosstable.gvl"
#import "Resource1.gvl"
CONST
	this : int := 16;
	test_cases : int := 7;
	xl : lreal := 0.0000000000000010;
	x : real :=   0.0000000000000001;
END_CONST
VAR
	test_case : array [1..test_cases] of lreal_lreal3_real3_T :=
[
(input:= -1.0000000000000000, retval1:=-1.5707963267948966, retval2:= 3.1415926535897931, retval3:=-0.7853981633974483, retval4:=-1.5707963267948966, retval5:= 3.1415926535897931, retval6:=-0.7853981633974483),
(input:= -0.6666666666666667, retval1:=-0.7297276562269664, retval2:= 2.3005239830218631, retval3:=-0.5880026035475676, retval4:=-0.7297276828829742, retval5:= 2.3005240096778707, retval6:=-0.5880026173024855),
(input:= -0.3333333333333334, retval1:=-0.3398369094541220, retval2:= 1.9106332362490186, retval3:=-0.3217505543966422, retval4:=-0.3398369199908341, retval5:= 1.9106332467857308, retval6:=-0.3217505633373389),
(input:=  0.0000000000000000, retval1:= 0.0000000000000000, retval2:= 1.5707963267948966, retval3:= 0.0000000000000000, retval4:= 0.0000000000000000, retval5:= 1.5707963267948966, retval6:= 0.0000000000000000),
(input:=  0.3333333333333333, retval1:= 0.3398369094541219, retval2:= 1.2309594173407747, retval3:= 0.3217505543966421, retval4:= 0.3398369199908341, retval5:= 1.2309594068040626, retval6:= 0.3217505633373389),
(input:=  0.6666666666666665, retval1:= 0.7297276562269661, retval2:= 0.8410686705679304, retval3:= 0.5880026035475675, retval4:= 0.7297276828829742, retval5:= 0.8410686439119225, retval6:= 0.5880026173024855),
(input:=  1.0000000000000000, retval1:= 1.5707963267948966, retval2:= 0.0000000000000000, retval3:= 0.7853981633974483, retval4:= 1.5707963267948966, retval5:= 0.0000000000000000, retval6:= 0.7853981633974483)
];
	input_lreal : lreal;
	input_real : real;
	retval1 : lreal;
	retval2 : lreal;
	retval3 : lreal;
	retval4 : real;
	retval5 : real;
	retval6 : real;

	index : int := 1;
	expected : string;
	obtained : string;
	result : bool;
END_VAR

	if Status = STATUS_RUNNING AND test_level_16 > TEST_DISABLED and test_loops_16 < Target then

		(* ---------- test action ---------------*)
		input_lreal := test_case[index].input;
        retval1 := asin(input_lreal);
        retval2 := acos(input_lreal);
        retval3 := atan(input_lreal);
		input_real := lreal_to_real(test_case[index].input);
        retval4 := asin(input_real);
        retval5 := acos(input_real);
        retval6 := atan(input_real);

		(* ---------- test condition ---------------*)
        result := (abs(retval1 - test_case[index].retval1) < xl)
		      and (abs(retval2 - test_case[index].retval2) < xl)
		      and (abs(retval3 - test_case[index].retval3) < xl)
		      and (abs(retval4 - test_case[index].retval4) < x)
		      and (abs(retval5 - test_case[index].retval5) < x)
		      and (abs(retval6 - test_case[index].retval6) < x);

		(* ---------- log message ---------------*)
		expected := '';
		expected := CONCAT(expected, comma_blank, lreal_to_string(test_case[index].retval1));
		expected := CONCAT(expected, comma_blank, lreal_to_string(test_case[index].retval2));
		expected := CONCAT(expected, comma_blank, lreal_to_string(test_case[index].retval3));
		expected := CONCAT(expected, comma_blank, real_to_string(test_case[index].retval4));
		expected := CONCAT(expected, comma_blank, real_to_string(test_case[index].retval5));
		expected := CONCAT(expected, comma_blank, real_to_string(test_case[index].retval6));
		obtained := '';
		obtained := CONCAT(obtained, comma_blank, lreal_to_string(retval1));
		obtained := CONCAT(obtained, comma_blank, lreal_to_string(retval2));
		obtained := CONCAT(obtained, comma_blank, lreal_to_string(retval3));
		obtained := CONCAT(obtained, comma_blank, real_to_string(retval4));
		obtained := CONCAT(obtained, comma_blank, real_to_string(retval5));
		obtained := CONCAT(obtained, comma_blank, real_to_string(retval6));

		(* ---------- cycle ----------*)
		SingleTest(this, result, expected, obtained, test_cases,
				   index, test_level_16, test_counter_16, test_loops_16, test_errors_16);
	end_if;
END_PROGRAM

(* ---- trig_P.st ---- *)
(*[[ ]]*)
PROGRAM trig_P
#import "Crosstable.gvl"
#import "Resource1.gvl"
CONST
	this : int := 15;
	test_cases : int := 7;
	xl : lreal := 0.0000000000000001;
	x : real := 0.0000000000000001;
END_CONST
VAR
	test_case : array [1..test_cases] of lreal_lreal3_real3_T :=
[
(input:= 0.0000000000000000, retval1:= 0.0000000000000000, retval2:= 1.0000000000000000, retval3:= 0.0000000000000000, retval4:= 0.0000000000000000, retval5:= 1.0000000000000000, retval6:= 0.0000000000000000),
(input:= 1.0471975511965976, retval1:= 0.8660254037844386, retval2:= 0.5000000000000001, retval3:= 1.7320508075688767, retval4:= 0.8660254183549017, retval5:= 0.4999999747632170, retval6:= 1.7320509241325899),
(input:= 2.0943951023931953, retval1:= 0.8660254037844387, retval2:=-0.4999999999999998, retval3:=-1.7320508075688783, retval4:= 0.8660253746435105, retval5:=-0.5000000504735648, retval6:=-1.7320505744414876),
(input:= 3.1415926535897931, retval1:= 0.0000000000000001, retval2:=-1.0000000000000000, retval3:=-0.0000000000000001, retval4:=-0.0000000874227800, retval5:=-0.9999999999999962, retval6:= 0.0000000874227800),
(input:= 4.1887902047863905, retval1:=-0.8660254037844384, retval2:=-0.5000000000000004, retval3:= 1.7320508075688754, retval4:=-0.8660254620662861, retval5:=-0.4999998990528655, retval6:= 1.7320512738237981),
(input:= 5.2359877559829879, retval1:=-0.8660254037844390, retval2:= 0.4999999999999993, retval3:=-1.7320508075688805, retval4:=-0.8660254501414079, retval5:= 0.4999999197073655, retval6:=-1.7320511784247199),
(input:= 6.2831853071795862, retval1:=-0.0000000000000002, retval2:= 1.0000000000000000, retval3:=-0.0000000000000002, retval4:= 0.0000001748455600, retval5:= 0.9999999999999847, retval6:= 0.0000001748455600)
];
	input_lreal : lreal;
	input_real : real;
	retval1 : lreal;
	retval2 : lreal;
	retval3 : lreal;
	retval4 : real;
	retval5 : real;
	retval6 : real;

	index : int := 1;
	expected : string;
	obtained : string;
	result : bool;
END_VAR

	if Status = STATUS_RUNNING AND test_level_15 > TEST_DISABLED and test_loops_15 < Target then

		(* ---------- test action ---------------*)
		input_lreal := test_case[index].input;
        retval1 := sin(input_lreal);
        retval2 := cos(input_lreal);
        retval3 := tan(input_lreal);
		input_real := lreal_to_real(test_case[index].input);
        retval4 := sin(input_real);
        retval5 := cos(input_real);
        retval6 := tan(input_real);

		(* ---------- test condition ---------------*)
        result := (abs(retval1 - test_case[index].retval1) < xl)
		      and (abs(retval2 - test_case[index].retval2) < xl)
		      and (abs(retval3 - test_case[index].retval3) < xl)
		      and (abs(retval4 - test_case[index].retval4) < x)
		      and (abs(retval5 - test_case[index].retval5) < x)
		      and (abs(retval6 - test_case[index].retval6) < x);

		(* ---------- log message ---------------*)
		expected := '';
		expected := CONCAT(expected, comma_blank, lreal_to_string(test_case[index].retval1));
		expected := CONCAT(expected, comma_blank, lreal_to_string(test_case[index].retval2));
		expected := CONCAT(expected, comma_blank, lreal_to_string(test_case[index].retval3));
		expected := CONCAT(expected, comma_blank, real_to_string(test_case[index].retval4));
		expected := CONCAT(expected, comma_blank, real_to_string(test_case[index].retval5));
		expected := CONCAT(expected, comma_blank, real_to_string(test_case[index].retval6));
		obtained := '';
		obtained := CONCAT(obtained, comma_blank, lreal_to_string(retval1));
		obtained := CONCAT(obtained, comma_blank, lreal_to_string(retval2));
		obtained := CONCAT(obtained, comma_blank, lreal_to_string(retval3));
		obtained := CONCAT(obtained, comma_blank, real_to_string(retval4));
		obtained := CONCAT(obtained, comma_blank, real_to_string(retval5));
		obtained := CONCAT(obtained, comma_blank, real_to_string(retval6));

		(* ---------- cycle ----------*)
		SingleTest(this, result, expected, obtained, test_cases,
				   index, test_level_15, test_counter_15, test_loops_15, test_errors_15);
	end_if;
END_PROGRAM

(* ---- trunc_P.st ---- *)
(*[[
]]*)
PROGRAM trunc_P
#import "Crosstable.gvl"
#import "Resource1.gvl"
CONST
	this : int := 10;
	test_cases : int := 5;
END_CONST
VAR
	test_case : array [1..test_cases] of lreal_any_int_T := [
		(input := -7.0, ret_int :=  -7, ret_dint := -7),
		(input := -2.2, ret_int :=  -2, ret_dint := -2),
		(input := 14.0, ret_int := 14, ret_dint := 14),
		(input := 14.11, ret_int := 14, ret_dint := 14),
		(input := 14.88, ret_int := 14, ret_dint := 14)
	];
	ret_int1  : int;
	ret_int2  : int;
	ret_dint1 : dint;
	ret_dint2 : dint;

	index : int := 1;
	expected : string;
	obtained : string;
	result : bool;
END_VAR

	if Status = STATUS_RUNNING AND test_level_10 > TEST_DISABLED and test_loops_10 < Target then

		(* ---------- test action ---------------*)
        ret_int1  := trunc(test_case[index].input);
        ret_dint1 := trunc(test_case[index].input);
        ret_int2  := trunc(lreal_to_real(test_case[index].input));
        ret_dint2 := trunc(lreal_to_real(test_case[index].input));

		(* ---------- test condition ---------------*)
        result := (ret_int1 = test_case[index].ret_int)
				  and (ret_dint1 = test_case[index].ret_dint)
				  and (ret_int2 = test_case[index].ret_int)
				  and (ret_dint2 = test_case[index].ret_dint);

		(* ---------- log message ---------------*)
		expected := '';
		expected := CONCAT(expected, comma_blank, int_to_string(test_case[index].ret_int));
		expected := CONCAT(expected, comma_blank, int_to_string(test_case[index].ret_int));
		expected := CONCAT(expected, comma_blank, dint_to_string(test_case[index].ret_dint));
		expected := CONCAT(expected, comma_blank, dint_to_string(test_case[index].ret_dint));
		obtained := '';
		obtained := CONCAT(obtained, comma_blank, int_to_string(ret_int1));
		obtained := CONCAT(obtained, comma_blank, int_to_string(ret_int2));
		obtained := CONCAT(obtained, comma_blank, dint_to_string(ret_dint1));
		obtained := CONCAT(obtained, comma_blank, dint_to_string(ret_dint2));

		(* ---------- cycle ----------*)
		SingleTest(this, result, expected, obtained, test_cases,
				   index, test_level_10, test_counter_10, test_loops_10, test_errors_10);
	end_if;

END_PROGRAM

(* ---- udint_to_all_P.st ---- *)
(*[[ ]]*)
PROGRAM udint_to_all_P
#import "Crosstable.gvl"
#import "Resource1.gvl"

CONST
	this : int := 11;
	test_cases : int := 4;
END_CONST
VAR
	test_case : array [1..test_cases] of udint_all_T := [
		(input := 0, ret_bool := 0, ret_byte := 0, ret_dint := 0, ret_dword := 0, ret_int := 0, ret_lreal := 0.0,
		   ret_real := 0.0, ret_string := '0', ret_word := 0),
		(input := 1, ret_bool := 1, ret_byte := 1, ret_dint := 1, ret_dword := 1, ret_int := 1, ret_lreal := 1.0,
		   ret_real := 1.0, ret_string := '1', ret_word := 1),
		(input := 255, ret_bool := 1, ret_byte := 255, ret_dint := 255, ret_dword := 255, ret_int := 255, ret_lreal := 255.0,
		   ret_real := 255.0, ret_string := '255', ret_word := 255),
		(input := 2559, ret_bool := 1, ret_byte := 255, ret_dint := 2559, ret_dword := 2559, ret_int := 2559, ret_lreal := 2559.0,
		   ret_real := 2559.0, ret_string := '2559', ret_word := 2559)
	];
    ret_bool   : bool;
    ret_byte   : byte;
    ret_dint   : dint;
    ret_dword  : dword;
    ret_int    : int;
    ret_lreal  : lreal;
    ret_real   : real;
    ret_string : string;
    ret_word   : word;

	index : int := 1;
	expected : string;
	obtained : string;
	result : bool;
END_VAR

	if Status = STATUS_RUNNING AND test_level_11 > TEST_DISABLED and test_loops_11 < Target then

		(* ---------- test action ---------------*)
        ret_bool   := udint_to_bool(test_case[index].input);
        ret_byte   := udint_to_byte(test_case[index].input);
        ret_dint   := udint_to_dint(test_case[index].input);
        ret_dword  := udint_to_dword(test_case[index].input);
        ret_int    := udint_to_int(test_case[index].input);
        ret_lreal  := udint_to_lreal(test_case[index].input);
        ret_real   := udint_to_real(test_case[index].input);
        ret_string := udint_to_string(test_case[index].input);
        ret_word   := udint_to_word(test_case[index].input);

		(* ---------- test condition ---------------*)
        result := (ret_bool = test_case[index].ret_bool)
		      and (ret_byte = test_case[index].ret_byte)
		      and (ret_dint = test_case[index].ret_dint)
		      and (ret_dword = test_case[index].ret_dword)
		      and (ret_int = test_case[index].ret_int)
		      and (ret_lreal = test_case[index].ret_lreal)
		      and (ret_real = test_case[index].ret_real)
		      and (ret_string = test_case[index].ret_string)
		      and (ret_word = test_case[index].ret_word);

		(* ---------- log message ---------------*)
		expected := '';
		expected := CONCAT(expected, comma_blank, bool_to_string(test_case[index].ret_bool));
		expected := CONCAT(expected, comma_blank, byte_to_string(test_case[index].ret_byte));
		expected := CONCAT(expected, comma_blank, dint_to_string(test_case[index].ret_dint));
		expected := CONCAT(expected, comma_blank, dword_to_string(test_case[index].ret_dword));
		expected := CONCAT(expected, comma_blank, int_to_string(test_case[index].ret_int));
		expected := CONCAT(expected, comma_blank, lreal_to_string(test_case[index].ret_lreal));
		expected := CONCAT(expected, comma_blank, real_to_string(test_case[index].ret_real));
		expected := CONCAT(expected, comma_blank, test_case[index].ret_string);
		expected := CONCAT(expected, comma_blank, word_to_string(test_case[index].ret_word));
		obtained := '';
		obtained := CONCAT(obtained, comma_blank, bool_to_string(ret_bool));
		obtained := CONCAT(obtained, comma_blank, byte_to_string(ret_byte));
		obtained := CONCAT(obtained, comma_blank, dint_to_string(ret_dint));
		obtained := CONCAT(obtained, comma_blank, dword_to_string(ret_dword));
		obtained := CONCAT(obtained, comma_blank, int_to_string(ret_int));
		obtained := CONCAT(obtained, comma_blank, lreal_to_string(ret_lreal));
		obtained := CONCAT(obtained, comma_blank, real_to_string(ret_real));
		obtained := CONCAT(obtained, comma_blank, ret_string);
		obtained := CONCAT(obtained, comma_blank, word_to_string(ret_word));

		(* ---------- cycle ----------*)
		SingleTest(this, result, expected, obtained, test_cases,
				   index, test_level_11, test_counter_11, test_loops_11, test_errors_11);
	end_if;
END_PROGRAM

(* ---- uint_to_all_P.st ---- *)
(*[[ ]]*)
PROGRAM uint_to_all_P
#import "Crosstable.gvl"
#import "Resource1.gvl"
CONST
	this : int := 12;
	test_cases : int := 4;
END_CONST
VAR
	test_case : array [1..test_cases] of uint_all_T := [
		(input := 0, ret_bool := 0, ret_byte := 0, ret_dint := 0, ret_dword := 0, ret_int := 0, ret_lreal := 0.0,
		   ret_real := 0.0, ret_string := '0', ret_word := 0),
		(input := 1, ret_bool := 1, ret_byte := 1, ret_dint := 1, ret_dword := 1, ret_int := 1, ret_lreal := 1.0,
		   ret_real := 1.0, ret_string := '1', ret_word := 1),
		(input := 255, ret_bool := 1, ret_byte := 255, ret_dint := 255, ret_dword := 255, ret_int := 255, ret_lreal := 255.0,
		   ret_real := 255.0, ret_string := '255', ret_word := 255),
		(input := 2559, ret_bool := 1, ret_byte := 255, ret_dint := 2559, ret_dword := 2559, ret_int := 2559, ret_lreal := 2559.0,
		   ret_real := 2559.0, ret_string := '2559', ret_word := 2559)
	];
    ret_bool   : bool;
    ret_byte   : byte;
    ret_dint   : dint;
    ret_dword  : dword;
    ret_int    : int;
    ret_lreal  : lreal;
    ret_real   : real;
    ret_string : string;
    ret_word   : word;

	index : int := 1;
	expected : string;
	obtained : string;
	result : bool;
END_VAR

	if Status = STATUS_RUNNING AND test_level_12 > TEST_DISABLED and test_loops_12 < Target then

		(* ---------- test action ---------------*)
        ret_bool   := uint_to_bool(test_case[index].input);
        ret_byte   := uint_to_byte(test_case[index].input);
        ret_dint   := uint_to_dint(test_case[index].input);
        ret_dword  := uint_to_dword(test_case[index].input);
        ret_int    := uint_to_int(test_case[index].input);
        ret_lreal  := uint_to_lreal(test_case[index].input);
        ret_real   := uint_to_real(test_case[index].input);
        ret_string := uint_to_string(test_case[index].input);
        ret_word   := uint_to_word(test_case[index].input);

		(* ---------- test condition ---------------*)
        result := (ret_bool = test_case[index].ret_bool)
		      and (ret_byte = test_case[index].ret_byte)
		      and (ret_dint = test_case[index].ret_dint)
		      and (ret_dword = test_case[index].ret_dword)
		      and (ret_int = test_case[index].ret_int)
		      and (ret_lreal = test_case[index].ret_lreal)
		      and (ret_real = test_case[index].ret_real)
		      and (ret_string = test_case[index].ret_string)
		      and (ret_word = test_case[index].ret_word);

		(* ---------- log message ---------------*)
		expected := '';
		expected := CONCAT(expected, comma_blank, bool_to_string(test_case[index].ret_bool));
		expected := CONCAT(expected, comma_blank, byte_to_string(test_case[index].ret_byte));
		expected := CONCAT(expected, comma_blank, dint_to_string(test_case[index].ret_dint));
		expected := CONCAT(expected, comma_blank, dword_to_string(test_case[index].ret_dword));
		expected := CONCAT(expected, comma_blank, int_to_string(test_case[index].ret_int));
		expected := CONCAT(expected, comma_blank, lreal_to_string(test_case[index].ret_lreal));
		expected := CONCAT(expected, comma_blank, real_to_string(test_case[index].ret_real));
		expected := CONCAT(expected, comma_blank, test_case[index].ret_string);
		expected := CONCAT(expected, comma_blank, word_to_string(test_case[index].ret_word));
		obtained := '';
		obtained := CONCAT(obtained, comma_blank, bool_to_string(ret_bool));
		obtained := CONCAT(obtained, comma_blank, byte_to_string(ret_byte));
		obtained := CONCAT(obtained, comma_blank, dint_to_string(ret_dint));
		obtained := CONCAT(obtained, comma_blank, dword_to_string(ret_dword));
		obtained := CONCAT(obtained, comma_blank, int_to_string(ret_int));
		obtained := CONCAT(obtained, comma_blank, lreal_to_string(ret_lreal));
		obtained := CONCAT(obtained, comma_blank, real_to_string(ret_real));
		obtained := CONCAT(obtained, comma_blank, ret_string);
		obtained := CONCAT(obtained, comma_blank, word_to_string(ret_word));

		(* ---------- cycle ----------*)
		SingleTest(this, result, expected, obtained, test_cases,
				   index, test_level_12, test_counter_12, test_loops_12, test_errors_12);
	end_if;
END_PROGRAM

(* ---- word_to_all_P.st ---- *)
(*[[ ]]*)
PROGRAM word_to_all_P
#import "Crosstable.gvl"
#import "Resource1.gvl"
CONST
	this : int := 13;
	test_cases : int := 4;
END_CONST
VAR
	test_case : array [1..test_cases] of word_all_T := [
		(input := 0, ret_bool := 0, ret_byte := 0, ret_dint := 0, ret_dword := 0, ret_int := 0, ret_lreal := 0.0,
		   ret_real := 0.0, ret_string := '0', ret_udint := 0, ret_uint := 0),
		(input := 1, ret_bool := 1, ret_byte := 1, ret_dint := 1, ret_dword := 1, ret_int := 1, ret_lreal := 1.0,
		   ret_real := 1.0, ret_string := '1', ret_udint := 1, ret_uint := 1),
		(input := 255, ret_bool := 1, ret_byte := 255, ret_dint := 255, ret_dword := 255, ret_int := 255, ret_lreal := 255.0,
		   ret_real := 255.0, ret_string := '255', ret_udint := 255, ret_uint := 255),
		(input := 2559, ret_bool := 1, ret_byte := 255, ret_dint := 2559, ret_dword := 2559, ret_int := 2559, ret_lreal := 2559.0,
		   ret_real := 2559.0, ret_string := '2559', ret_udint := 2559, ret_uint := 2559)
	];
    ret_bool   : bool;
    ret_byte   : byte;
    ret_dint   : dint;
    ret_dword  : dword;
    ret_int    : int;
    ret_lreal  : lreal;
    ret_real   : real;
    ret_string : string;
    ret_udint  : udint;
    ret_uint   : uint;

	index : int := 1;
	expected : string;
	obtained : string;
	result : bool;
END_VAR

	if Status = STATUS_RUNNING AND test_level_13 > TEST_DISABLED and test_loops_13 < Target then

		(* ---------- test action ---------------*)
        ret_bool   := word_to_bool(test_case[index].input);
        ret_byte   := word_to_byte(test_case[index].input);
        ret_dint   := word_to_dint(test_case[index].input);
        ret_dword  := word_to_dword(test_case[index].input);
        ret_int    := word_to_int(test_case[index].input);
        ret_lreal  := word_to_lreal(test_case[index].input);
        ret_real   := word_to_real(test_case[index].input);
        ret_string := word_to_string(test_case[index].input);
        ret_udint  := word_to_udint(test_case[index].input);
        ret_uint   := word_to_uint(test_case[index].input);

		(* ---------- test condition ---------------*)
        result := (ret_bool = test_case[index].ret_bool)
		      and (ret_byte = test_case[index].ret_byte)
		      and (ret_dint = test_case[index].ret_dint)
		      and (ret_dword = test_case[index].ret_dword)
		      and (ret_int = test_case[index].ret_int)
		      and (ret_lreal = test_case[index].ret_lreal)
		      and (ret_real = test_case[index].ret_real)
		      and (ret_string = test_case[index].ret_string)
		      and (ret_udint = test_case[index].ret_udint)
		      and (ret_uint = test_case[index].ret_uint);

		(* ---------- log message ---------------*)
		expected := '';
		expected := CONCAT(expected, comma_blank, bool_to_string(test_case[index].ret_bool));
		expected := CONCAT(expected, comma_blank, byte_to_string(test_case[index].ret_byte));
		expected := CONCAT(expected, comma_blank, dint_to_string(test_case[index].ret_dint));
		expected := CONCAT(expected, comma_blank, dword_to_string(test_case[index].ret_dword));
		expected := CONCAT(expected, comma_blank, int_to_string(test_case[index].ret_int));
		expected := CONCAT(expected, comma_blank, lreal_to_string(test_case[index].ret_lreal));
		expected := CONCAT(expected, comma_blank, real_to_string(test_case[index].ret_real));
		expected := CONCAT(expected, comma_blank, test_case[index].ret_string);
		expected := CONCAT(expected, comma_blank, udint_to_string(test_case[index].ret_udint));
		expected := CONCAT(expected, comma_blank, uint_to_string(test_case[index].ret_uint));
		obtained := '';
		obtained := CONCAT(obtained, comma_blank, bool_to_string(ret_bool));
		obtained := CONCAT(obtained, comma_blank, byte_to_string(ret_byte));
		obtained := CONCAT(obtained, comma_blank, dint_to_string(ret_dint));
		obtained := CONCAT(obtained, comma_blank, dword_to_string(ret_dword));
		obtained := CONCAT(obtained, comma_blank, int_to_string(ret_int));
		obtained := CONCAT(obtained, comma_blank, lreal_to_string(ret_lreal));
		obtained := CONCAT(obtained, comma_blank, real_to_string(ret_real));
		obtained := CONCAT(obtained, comma_blank, ret_string);
		obtained := CONCAT(obtained, comma_blank, udint_to_string(ret_udint));
		obtained := CONCAT(obtained, comma_blank, uint_to_string(ret_uint));

		(* ---------- cycle ----------*)
		SingleTest(this, result, expected, obtained, test_cases,
				   index, test_level_13, test_counter_13, test_loops_13, test_errors_13);
	end_if;
END_PROGRAM

(* ---- xor_P.st ---- *)
(*[[ ]]*)
PROGRAM xor_P
#import "Crosstable.gvl"
#import "Resource1.gvl"
CONST
	this : int := 30;
	test_cases : int := 13;
END_CONST
VAR
	test_case : array [1..test_cases] of bit2_bit_T := [
		(input0 := 0, 		    input1 := 0, 	 	   ret_bool := 0, ret_byte := 0, 	 ret_word := 0, 	ret_dword := 0),
		(input0 := 0, 			input1 := 1, 	   	   ret_bool := 1, ret_byte := 1, 	 ret_word := 1, 	ret_dword := 1),
		(input0 := 1, 			input1 := 0, 	   	   ret_bool := 1, ret_byte := 1, 	 ret_word := 1, 	ret_dword := 1),
		(input0 := 1, 			input1 := 1, 	       ret_bool := 0, ret_byte := 0, 	 ret_word := 0, 	ret_dword := 0),
		(input0 := 0, 			input1 := 16#000000ff, ret_bool := 1, ret_byte := 16#ff, ret_word := 16#00ff, ret_dword := 16#000000ff),
		(input0 := 16#000000ff, input1 := 16#000000ff, ret_bool := 0, ret_byte := 16#00, ret_word := 16#0000, ret_dword := 16#00000000),
		(input0 := 16#0000000f, input1 := 16#000000f0, ret_bool := 0, ret_byte := 16#ff, ret_word := 16#00ff, ret_dword := 16#000000ff),
		(input0 := 16#0000ffff, input1 := 16#0000ffff, ret_bool := 0, ret_byte := 16#00, ret_word := 16#0000, ret_dword := 16#00000000),
		(input0 := 16#0000ffff, input1 := 16#000000ff, ret_bool := 0, ret_byte := 16#00, ret_word := 16#ff00, ret_dword := 16#0000ff00),
		(input0 := 16#0000f000, input1 := 16#0000ffff, ret_bool := 0, ret_byte := 16#ff, ret_word := 16#0fff, ret_dword := 16#00000fff),
		(input0 := 16#000000ff, input1 := 16#0000ff00, ret_bool := 0, ret_byte := 16#ff, ret_word := 16#ffff, ret_dword := 16#0000ffff),
		(input0 := 16#abcde012, input1 := 16#ffffffff, ret_bool := 0, ret_byte := 16#ed, ret_word := 16#1fed, ret_dword := 16#54321fed),
		(input0 := 16#abcdefab, input1 := 16#ff000000, ret_bool := 0, ret_byte := 16#ab, ret_word := 16#efab, ret_dword := 16#54cdefab)
	];
    ret_bool   : bool;
    ret_byte   : byte;
    ret_word   : word;
    ret_dword  : dword;

	index : int := 1;
	expected : string;
	obtained : string;
	result : bool;
END_VAR

	if Status = STATUS_RUNNING AND test_level_30 > TEST_DISABLED and test_loops_30 < Target then

		(* ---------- test action ---------------*)
        ret_bool   := xor(dword_to_bool(test_case[index].input0), dword_to_bool(test_case[index].input1));
        ret_byte   := xor(dword_to_byte(test_case[index].input0), dword_to_byte(test_case[index].input1));
        ret_word   := xor(dword_to_word(test_case[index].input0), dword_to_word(test_case[index].input1));
        ret_dword  := xor(test_case[index].input0, test_case[index].input1);

		(* ---------- test condition ---------------*)
        result := (ret_bool = test_case[index].ret_bool)
		      and (ret_byte = test_case[index].ret_byte)
		      and (ret_word = test_case[index].ret_word)
		      and (ret_dword = test_case[index].ret_dword);

		(* ---------- log message ---------------*)
		expected := '';
		expected := CONCAT(expected, comma_blank, bool_to_string(test_case[index].ret_bool));
		expected := CONCAT(expected, comma_blank, byte_to_string(test_case[index].ret_byte));
		expected := CONCAT(expected, comma_blank, word_to_string(test_case[index].ret_word));
		expected := CONCAT(expected, comma_blank, dword_to_string(test_case[index].ret_dword));
		obtained := '';
		obtained := CONCAT(obtained, comma_blank, bool_to_string(ret_bool));
		obtained := CONCAT(obtained, comma_blank, byte_to_string(ret_byte));
		obtained := CONCAT(obtained, comma_blank, word_to_string(ret_word));
		obtained := CONCAT(obtained, comma_blank, dword_to_string(ret_dword));

		(* ---------- cycle ----------*)
		SingleTest(this, result, expected, obtained, test_cases,
				   index, test_level_30, test_counter_30, test_loops_30, test_errors_30);
	end_if;
END_PROGRAM

(* ---- xx_no_test_P.st ---- *)
(*[[
]]*)
PROGRAM xx_no_test_P
VAR
END_VAR

;
END_PROGRAM

(* ---- xx_TestInit.st ---- *)
(*[[
]]*)
PROGRAM xx_TestInit
#import "Crosstable.gvl"
#import "Resource1.gvl"

	SetDefaultValues();
	ResetCounters();
	UpdateCounters();

	Status := STATUS_IDLE;

END_PROGRAM

(* ---- xx_TestManager.st ---- *)
(*[[
]]*)
PROGRAM xx_TestManager
#import "Crosstable.gvl"
#import "Resource1.gvl"
VAR
	StartTime_cs : UDINT := 0;
END_VAR

	case Status of

	STATUS_ZERO:
		;

	STATUS_IDLE:
		if BUTTON_START then
			StartTest();
			StartTime_cs := PLC_UPTIME_cs;
			Elapsed_s := 0;
			Status := STATUS_RUNNING;
		elsif BUTTON_RESET then
			SetDefaultValues();
			ResetCounters();
			UpdateCounters();
		else
			;
		end_if;

	STATUS_RUNNING:
		UpdateCounters();
		if BUTTON_STOP then
			StopTest();
			Status := STATUS_DONE;
		else
			Elapsed_s := PLC_UPTIME_cs - StartTime_cs; (* NB: Elapsed_s has decimals = 2 *)
			StepTest();
			if Target > 0 and Loops >= Target then
				StopTest();
				Status := STATUS_DONE;
			end_if;
		end_if;

	STATUS_DONE:
		if BUTTON_START then
			ResetCounters();
			UpdateCounters();
			StartTest();
			StartTime_cs := PLC_UPTIME_cs;
			Elapsed_s := 0;
			Status := STATUS_RUNNING;
		elsif BUTTON_RESET then
			SetDefaultValues();
			ResetCounters();
			UpdateCounters();
			Status := STATUS_IDLE;
		else
			;
		end_if;

	else
		;

	end_case;

END_PROGRAM

(* ---- xx_TestMonitor.st ---- *)
(*[[
]]*)
PROGRAM xx_TestMonitor
#import "Crosstable.gvl"
#import "Resource1.gvl"
VAR
	stat  : TSK_STAT;
	retval : word;
END_VAR

	retval := TSK_GetStatistic('Task00_TestInit'        , stat);	ETMAX_Task00 := stat.ExecMax;	ETAVG_Task00 := stat.ExecAverage;
	retval := TSK_GetStatistic('Task01_TestManager'     , stat);	ETMAX_Task01 := stat.ExecMax;	ETAVG_Task01 := stat.ExecAverage;
	retval := TSK_GetStatistic('Task02_TestMonitor'     , stat);	ETMAX_Task02 := stat.ExecMax;	ETAVG_Task02 := stat.ExecAverage;

	retval := TSK_GetStatistic('Task03_ATCM_File'       , stat);	ETMAX_Task03 := stat.ExecMax;	ETAVG_Task03 := stat.ExecAverage;
	retval := TSK_GetStatistic('Task04_ATCM_IEC1131_3_A', stat);	ETMAX_Task04 := stat.ExecMax;	ETAVG_Task04 := stat.ExecAverage;
	retval := TSK_GetStatistic('Task05_ATCM_IEC1131_3_B', stat);	ETMAX_Task05 := stat.ExecMax;	ETAVG_Task05 := stat.ExecAverage;
	retval := TSK_GetStatistic('Task06_ATCM_IEC1131_3_C', stat);	ETMAX_Task06 := stat.ExecMax;	ETAVG_Task06 := stat.ExecAverage;
	retval := TSK_GetStatistic('Task07_ATCM_IEC1131_3_D', stat);	ETMAX_Task07 := stat.ExecMax;	ETAVG_Task07 := stat.ExecAverage;
	retval := TSK_GetStatistic('Task08_ATCM_IEC1131_3_E', stat);	ETMAX_Task08 := stat.ExecMax;	ETAVG_Task08 := stat.ExecAverage;
	retval := TSK_GetStatistic('Task09_ATCM_IEC1131_3_F', stat);	ETMAX_Task09 := stat.ExecMax;	ETAVG_Task09 := stat.ExecAverage;
	retval := TSK_GetStatistic('Task10_ATCM_IEC1131_3_G', stat);	ETMAX_Task10 := stat.ExecMax;	ETAVG_Task10 := stat.ExecAverage;
	retval := TSK_GetStatistic('Task11_ATCM_IEC1131_3_H', stat);	ETMAX_Task11 := stat.ExecMax;	ETAVG_Task11 := stat.ExecAverage;
	retval := TSK_GetStatistic('Task12_ATCM_IEC1131_3_I', stat);	ETMAX_Task12 := stat.ExecMax;	ETAVG_Task12 := stat.ExecAverage;
	retval := TSK_GetStatistic('Task13_ATCM_IEC1131_3_J', stat);	ETMAX_Task13 := stat.ExecMax;	ETAVG_Task13 := stat.ExecAverage;
	retval := TSK_GetStatistic('Task14_ATCM_IEC1131_3_K', stat);	ETMAX_Task14 := stat.ExecMax;	ETAVG_Task14 := stat.ExecAverage;
	retval := TSK_GetStatistic('Task15_ATCM_IEC1131_3_L', stat);	ETMAX_Task15 := stat.ExecMax;	ETAVG_Task15 := stat.ExecAverage;
	retval := TSK_GetStatistic('Task16_ATCM_IEC1131_3_M', stat);	ETMAX_Task16 := stat.ExecMax;	ETAVG_Task16 := stat.ExecAverage;
	retval := TSK_GetStatistic('Task17_ATCM_System'     , stat);	ETMAX_Task17 := stat.ExecMax;	ETAVG_Task17 := stat.ExecAverage;
	retval := TSK_GetStatistic('Task18_ATCM_System2'    , stat);	ETMAX_Task18 := stat.ExecMax;	ETAVG_Task18 := stat.ExecAverage;
	retval := TSK_GetStatistic('Task19_ATCM_Utility'    , stat);	ETMAX_Task19 := stat.ExecMax;	ETAVG_Task19 := stat.ExecAverage;

END_PROGRAM
